ABB RobotStudio station: ABB_Pick&Place_v1.0_20230122-001637.rsstn

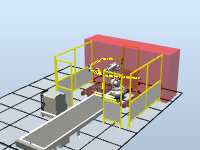
Station ABB_Pick&Place_v1.0 (saved by RobotStudio 6.8.8307.1040)
Controller Controller_Pick_Place_1, task T_ROB1: task frame (RAPID world) sits at (4966, 0, 259) mm, rotated rx 0 ry 0 rz 180 deg in the station
Controller Controller_Pick_Place_1
  mechanical unit ROB_1: IRB1660ID_4_155__03, 6 joints, base frame (0, 0, 0) mm
Layout (positions relative to the parent item):
  - 950_4000_h2 [part, from Equipment\Conveyor 950 4000 h2.rslib] at (0, -475, 0) mm
  - SC_Conveyor [smart component]
      signals: DI Crear_Caja_pq, DI Crear_Caja_gr, DO DO_Sensor_Sup, DO DO_Sensor_Inf
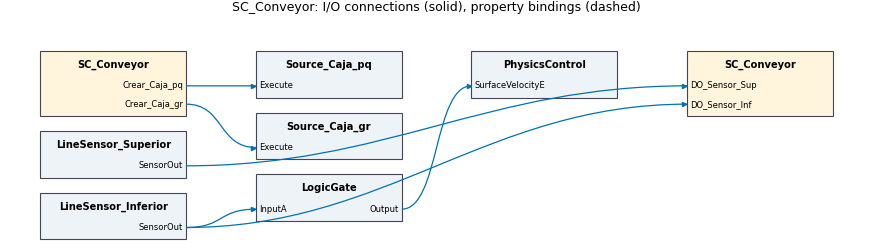
      connections:
        SC_Conveyor.Crear_Caja_pq -> Source_Caja_pq.Execute
        SC_Conveyor.Crear_Caja_gr -> Source_Caja_gr.Execute
        LineSensor_Superior.SensorOut -> SC_Conveyor.DO_Sensor_Sup
        LineSensor_Inferior.SensorOut -> SC_Conveyor.DO_Sensor_Inf
        LineSensor_Inferior.SensorOut -> LogicGate.InputA
        LogicGate.Output -> PhysicsControl.SurfaceVelocityEnabled
    - Caja_gr [part] at (85, -100, 680) mm
    - Caja_pq [part] at (85, -100, 580) mm
    - Cinta [part] at (60, -475, 375) mm
    - Source_Caja_pq [smart component, from Components\Source.rslib]
        properties: Source=Caja_pq; Copy=(none); Parent=(none); Position=[0.085 -0.1 0.58]; Orientation=[0 0 0]; Transient=true; PhysicsBehavior=3
    - Source_Caja_gr [smart component, from Components\Source.rslib]
        properties: Source=Caja_gr; Copy=(none); Parent=(none); Position=[0.085 -0.1 0.68]; Orientation=[0 0 0]; Transient=true; PhysicsBehavior=3
    - PhysicsControl [smart component, from Components\PhysicsControl.rslib]
        properties: Object=Cinta; Behavior=1; SurfaceVelocity=0.4
    - LineSensor_Inferior [smart component, from Components\LineSensor.rslib]
        properties: Start=[4 0.435 0.465]; End=[4 -0.475 0.465]; Radius=0; SensedPart=(none); SensedPoint=[0 0 0]
      - _sensorPart_ [part]
    - LineSensor_Superior [smart component, from Components\LineSensor.rslib]
        properties: Start=[4 0.435 0.565]; End=[4 -0.475 0.565]; Radius=0; SensedPart=(none); SensedPoint=[0 0 0]
      - _sensorPart_ [part]
    - LogicGate [smart component, from Components\LogicGate.rslib]
        properties: Operator=NOT; Delay=0
  - Robotpedestal1400_H240 [part, from Equipment\Robot Pedestal 1400 H240.rslib] at (5000, 0, 0) mm
  - IRB1660ID_4_155__03 [mechanism, from Robots\IRB1660ID_4_155__03.rslib] at (4966, 0, 259) mm, rotated rx 0 ry 0 rz 180 deg; joint values [0, 0, 0, 0, 0.5236, 0] (rad or m)
  - SC_VentosaTool [smart component] at (4021.13, 0, 1488) mm, rotated rx -180 ry 60 rz 0 deg
      signals: DI DI_Attach
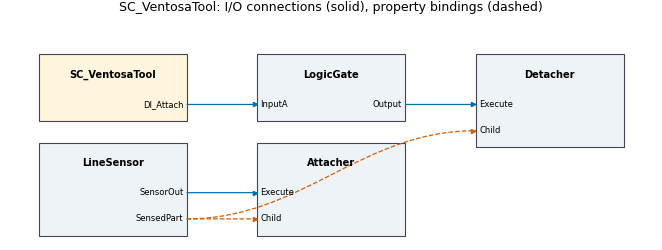
      connections:
        SC_VentosaTool.DI_Attach -> LogicGate.InputA
        LogicGate.Output -> Detacher.Execute
        LineSensor.SensorOut -> Attacher.Execute
        LineSensor.SensedPart => Attacher.Child
        LineSensor.SensedPart => Detacher.Child
    - VentosaTool [mechanism, from Libraries\VentosaTool.rslib] at (0, 0, 0) mm
    - Attacher [smart component, from Components\Attacher.rslib]
        properties: Parent=VentosaTool; Flange=0; Child=(none); Mount=false; Offset=[0 0 0]; Orientation=[0 0 0]
    - Detacher [smart component, from Components\Detacher.rslib]
        properties: Child=(none); KeepPosition=true
    - LogicGate [smart component, from Components\LogicGate.rslib]
        properties: Operator=NOT; Delay=0
    - LineSensor [smart component, from Components\LineSensor.rslib]
        properties: Start=[0 0 0.18]; End=[0 0 0.2]; Radius=0.001; SensedPart=(none); SensedPoint=[0 0 0]
      - _sensorPart_ [part]
  - IRC5_Singel-Cabinet [part, from Equipment\IRC5_Singel-Cabinet.rslib] at (2260, 1160, 100) mm, rotated rx 90 ry 0 rz -90 deg
  - Euro Pallet [graphiccomponentgroup, from Equipment\Euro Pallet.rslib] at (4400, -1365, 0) mm
    - Body 1 [part, from Equipment\Euro Pallet.rslib]
  - Euro Pallet_2 [graphiccomponentgroup, from Equipment\Euro Pallet.rslib] at (4444, 650, 0) mm
    - Body 1 [part, from Equipment\Euro Pallet.rslib]
  - Caja_gr_2 [part] at (4925, -1070, 144) mm
  - Caja_pq_2 [part] at (4950, 940, 144) mm
  - Fence_740 [graphiccomponentgroup, from Equipment\Fence_740.rslib] at (3000, 750, 0) mm
    - Body 1 [part, from Equipment\Fence_740.rslib]
    - Body 2 [part, from Equipment\Fence_740.rslib]
  - Fence_740_2 [graphiccomponentgroup, from Equipment\Fence_740.rslib] at (3000, -1350, 0) mm
    - Body 1 [part, from Equipment\Fence_740.rslib]
    - Body 2 [part, from Equipment\Fence_740.rslib]
  - Fence_2500 [graphiccomponentgroup, from Equipment\Fence_2500.rslib] at (5712, 1734, 0) mm, rotated rx 0 ry 0 rz 90 deg
    - Body 1 [part, from Equipment\Fence_2500.rslib]
    - Body 2 [part, from Equipment\Fence_2500.rslib]
  - Fence_2500_2 [graphiccomponentgroup, from Equipment\Fence_2500.rslib] at (5713, -1550, 0) mm, rotated rx 0 ry 0 rz 90 deg
    - Body 1 [part, from Equipment\Fence_2500.rslib]
    - Body 2 [part, from Equipment\Fence_2500.rslib]
  - Fence_740_3 [graphiccomponentgroup, from Equipment\Fence_740.rslib] at (6000, -370, 0) mm
    - Body 1 [part, from Equipment\Fence_740.rslib]
    - Body 2 [part, from Equipment\Fence_740.rslib]
  - Assem EMERGENCY PUSH BUTTON AND SWETSH OUTDOOR [part] at (2945, -1340, 950) mm, rotated rx 90 ry 0 rz -90 deg
  - Assem EMERGENCY PUSH BUTTON AND SWETSH OUTDOOR_2 [part] at (6053, -360, 950) mm, rotated rx 90 ry 0 rz 90 deg
  - COLUNA LUMINOSA [part] at (2994, -1355, 1993) mm, rotated rx 90 ry 0 rz 0 deg
  - MS4800B_30_[]_SIDEMOUNT_2 [part] at (5765, 1733, 400) mm, rotated rx 90 ry 0 rz 0 deg
  - MS4800B_30_[]_SIDEMOUNT_3 [part] at (5765, -1547, 400) mm, rotated rx 90 ry 0 rz 0 deg
  - WorldZone [part] at (5700, -1860, 0) mm
Attachment: SC_VentosaTool is attached to IRB1660ID_4_155__03 / Link6
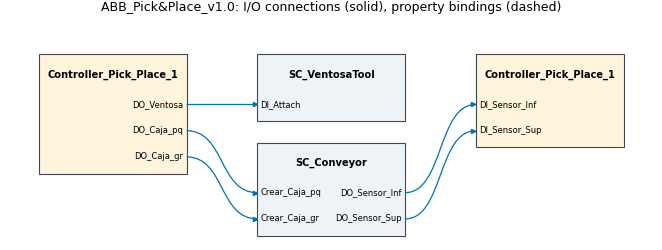
Station logic (signal -> signal, property => property):
  SC_Conveyor.DO_Sensor_Inf -> Controller_Pick_Place_1.DI_Sensor_Inf
  SC_Conveyor.DO_Sensor_Sup -> Controller_Pick_Place_1.DI_Sensor_Sup
  Controller_Pick_Place_1.DO_Ventosa -> SC_VentosaTool.DI_Attach
  Controller_Pick_Place_1.DO_Caja_pq -> SC_Conveyor.Crear_Caja_pq
  Controller_Pick_Place_1.DO_Caja_gr -> SC_Conveyor.Crear_Caja_gr
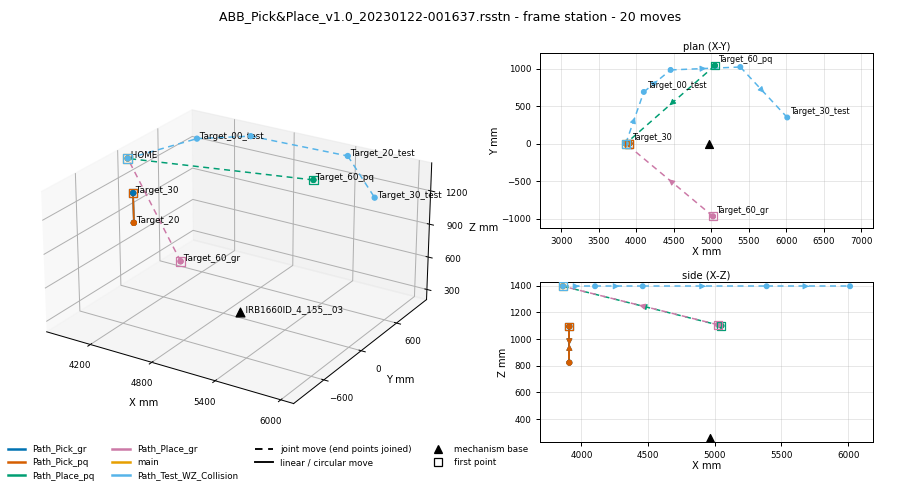
[picture p0: tool path of ABB_Pick&Place_v1.0_20230122-001637.rsstn in frame station, 20 of 24 moves have a stored position in this frame; points joined in program order, loops and branches not executed]
Targets, tools, work objects and paths stored in the station, written as RAPID:
! task T_ROB1
MODULE CalibData
  PERS tooldata TCP_VentosaTool:=[TRUE,[[0,0,184],[1,0,0,0]],[1,[0,-0.818,79.529],[1,0,0,0],0,0,0]];
  TASK PERS wobjdata WO_Pick:=[FALSE,TRUE,"",[[846,535,176],[1,0,0,0]],[[0,0,0],[1,0,0,0]]];
  TASK PERS wobjdata WO_Place_pq:=[FALSE,TRUE,"",[[522,-650,-259],[1,0,0,0]],[[0,0,0],[1,0,0,0]]];
  TASK PERS wobjdata WO_Place_gr:=[FALSE,TRUE,"",[[566,1365,-259],[1,0,0,0]],[[0,0,0],[1,0,0,0]]];
ENDMODULE

! task T_ROB1
MODULE Module1
  CONST robtarget HOME:=[[1104.222103807,0,1137],[0.5,0,0.866025404,0],[0,0,0,0],[9E+09,9E+09,9E+09,9E+09,9E+09,9E+09]];
  CONST robtarget Target_10_Pick_gr:=[[210.484,-535.003,180],[0,0,1,0],[0,0,0,0],[9E+09,9E+09,9E+09,9E+09,9E+09,9E+09]];
  CONST robtarget Target_20:=[[210.484,-535.003,388.047028658],[0,0,1,0],[0,0,0,0],[9E+09,9E+09,9E+09,9E+09,9E+09,9E+09]];
  CONST robtarget Target_30:=[[210.484,-535.003,659.509563159],[0,0,1,0],[0,0,0,0],[9E+09,9E+09,9E+09,9E+09,9E+09,9E+09]];
  CONST robtarget Target_10_Pick_pq:=[[210.488,-535,80],[0,0,1,0],[0,0,0,0],[9E+09,9E+09,9E+09,9E+09,9E+09,9E+09]];
  CONST robtarget Target_40_Place_pq:=[[-606,-390,244],[0,0.707106781,0.707106781,0],[-2,0,-1,0],[9E+09,9E+09,9E+09,9E+09,9E+09,9E+09]];
  CONST robtarget Target_50_pq:=[[-606,-390,486.324432044],[0,0.707106781,0.707106781,0],[-2,0,-1,0],[9E+09,9E+09,9E+09,9E+09,9E+09,9E+09]];
  CONST robtarget Target_60_pq:=[[-606,-390,1099.439558744],[0,0.707106781,0.707106781,0],[-2,0,-1,0],[9E+09,9E+09,9E+09,9E+09,9E+09,9E+09]];
  CONST robtarget Target_40_Place_gr:=[[-625,-395,344],[0,-0.707106781,0.707106781,0],[0,0,0,0],[9E+09,9E+09,9E+09,9E+09,9E+09,9E+09]];
  CONST robtarget Target_50_gr:=[[-625,-395,582.196057738],[0,-0.707106781,0.707106781,0],[0,0,0,0],[9E+09,9E+09,9E+09,9E+09,9E+09,9E+09]];
  CONST robtarget Target_60_gr:=[[-625,-395,1107.166955268],[0,-0.707106781,0.707106781,0],[0,0,0,0],[9E+09,9E+09,9E+09,9E+09,9E+09,9E+09]];
  CONST robtarget Target_10_test:=[[506.226977226,-981.346320927,1137.000114297],[0.426972887,0.45064673,0.739538717,-0.260181022],[-1,0,-1,0],[9E+09,9E+09,9E+09,9E+09,9E+09,9E+09]];
  CONST robtarget Target_30_test:=[[-1048.084035334,-347.600645778,1137.000114297],[0.079717809,0.854947485,0.138075298,-0.493604175],[-2,0,-1,0],[9E+09,9E+09,9E+09,9E+09,9E+09,9E+09]];
  CONST robtarget Target_20_test:=[[-422.599832723,-1020.154776185,1136.999978871],[0.277778532,0.720081419,0.481126538,-0.415739211],[-2,0,-1,0],[9E+09,9E+09,9E+09,9E+09,9E+09,9E+09]];
  CONST robtarget Target_00_test:=[[863.651388816,-688.049895242,1136.999985424],[0.471981945,0.285830632,0.817496693,-0.165024395],[-1,0,-1,0],[9E+09,9E+09,9E+09,9E+09,9E+09,9E+09]];
  PROC Path_Pick_gr()
    MoveJ Target_30,v1000,z100,TCP_VentosaTool\WObj:=WO_Pick;
    MoveL Target_20,v1000,z100,TCP_VentosaTool\WObj:=WO_Pick;
    WaitTime 1;
    MoveL Target_20,v1000,z100,TCP_VentosaTool\WObj:=WO_Pick;
    MoveL Target_30,v1000,z100,TCP_VentosaTool\WObj:=WO_Pick;
  ENDPROC
  PROC Path_Pick_pq()
    MoveJ Target_30,v1000,z100,TCP_VentosaTool\WObj:=WO_Pick;
    MoveL Target_20,v1000,z100,TCP_VentosaTool\WObj:=WO_Pick;
    WaitTime 1;
    MoveL Target_20,v1000,z100,TCP_VentosaTool\WObj:=WO_Pick;
    MoveL Target_30,v1000,z100,TCP_VentosaTool\WObj:=WO_Pick;
  ENDPROC
  PROC Path_Place_pq()
    MoveJ Target_60_pq,v1000,z100,TCP_VentosaTool\WObj:=WO_Place_pq;
    MoveL offs(Target_50_pq,0,0,off_pq),v1000,z100,TCP_VentosaTool\WObj:=WO_Place_pq;
    WaitTime 1;
    MoveL offs(Target_50_pq,0,0,off_pq),v1000,z100,TCP_VentosaTool\WObj:=WO_Place_pq;
    MoveL Target_60_pq,v1000,z100,TCP_VentosaTool\WObj:=WO_Place_pq;
    MoveJ HOME,v1000,z100,TCP_VentosaTool\WObj:=wobj0;
  ENDPROC
  PROC Path_Place_gr()
    MoveJ Target_60_gr,v1000,z100,TCP_VentosaTool\WObj:=WO_Place_gr;
    MoveL offs(Target_50_gr,0,0,off_gr),v1000,z100,TCP_VentosaTool\WObj:=WO_Place_gr;
    WaitTime 1;
    MoveL offs(Target_50_gr,0,0,off_gr),v1000,z100,TCP_VentosaTool\WObj:=WO_Place_gr;
    MoveL Target_60_gr,v1000,z100,TCP_VentosaTool\WObj:=WO_Place_gr;
    MoveJ HOME,v1000,z100,TCP_VentosaTool\WObj:=wobj0;
  ENDPROC
  PROC main()
    MoveJ HOME,v1000,z100,TCP_VentosaTool\WObj:=wobj0;
    create_box;
    PathCaja_pq;
    PathCaja_gr;
  ENDPROC
  PROC create_box()
    Set DO_Caja_pq;
    WaitTime 2;
    Reset DO_Caja_pq;
    Set DO_Caja_gr;
    WaitTime 2;
    Reset DO_Caja_gr;
  ENDPROC
  PROC PathCaja_gr()
    Path_Pick_gr;
    Path_Place_gr;
  ENDPROC
  PROC PathCaja_pq()
    Path_Pick_pq;
    Path_Place_pq;
  ENDPROC
  PROC Path_Test_WZ_Collision()
    MoveJ HOME,v500,z100,TCP_VentosaTool\WObj:=wobj0;
    MoveJ Target_00_test,v1000,z100,TCP_VentosaTool\WObj:=wobj0;
    MoveJ Target_10_test,v1000,z100,TCP_VentosaTool\WObj:=wobj0;
    MoveJ Target_20_test,v500,z100,TCP_VentosaTool\WObj:=wobj0;
    MoveJ Target_30_test,v500,z100,TCP_VentosaTool\WObj:=wobj0;
  ENDPROC
ENDMODULE

